// TIA Portal V18 export
// export: Created 2025-12-01T12:38:51.9439054Z, ExportSetting None, DisplayName Totally Integrated Automation Portal, DisplayVersion V18 Update 5, DisplayName TIA Portal Openness, DisplayVersion V18 Update 5, DisplayName TIA Portal Teamcenter Gateway, DisplayVersion V18, DisplayName TIA Portal Version Control Interface, DisplayVersion V18, DisplayName STEP 7 Professional, DisplayVersion V18 Update 5, DisplayName STEP 7 Safety, DisplayVersion V18, DisplayName WinCC Professional, DisplayVersion V18 Update 5
DATA_BLOCK "MES_CheckControl"   // DB2361
{ S7_Optimized_Access := 'FALSE' }
// stored: AutoNumber false
   VAR
      ST1MesCheckIn : Bool;
      ST1MesCheckOut : Bool;
      ST2MesCheckIn : Bool;
      ST2MesCheckOut : Bool;
      ST3MesCheckIn : Bool;
      ST3MesCheckOut : Bool;
      ST4MesCheckIn : Bool;
      ST4MesCheckOut : Bool;
      Station1 : Struct
         CheckInRequest : Bool;
         CheckResultRequest : Bool;
      END_STRUCT;
      Station2 : Struct
         CheckInRequest : Bool;
         CheckResultRequest : Bool;
      END_STRUCT;
      Station3 : Struct
         CheckInRequest : Bool;
         CheckResultRequest : Bool;
      END_STRUCT;
      Station4 : Struct
         CheckInRequest : Bool;
         CheckResultRequest : Bool;
      END_STRUCT;
      Station5 : Struct
         CheckInRequest : Bool;
         CheckResultRequest : Bool;
      END_STRUCT;
      Station6 : Struct
         CheckInRequest : Bool;
         CheckResultRequest : Bool;
      END_STRUCT;
      Station7 : Struct
         CheckInRequest : Bool;
         CheckResultRequest : Bool;
      END_STRUCT;
   END_VAR
BEGIN
END_DATA_BLOCK
